// Mitsubishi GX Works2 project: mc_protocol   PLC: Q03UDV

PROGRAM MAIN
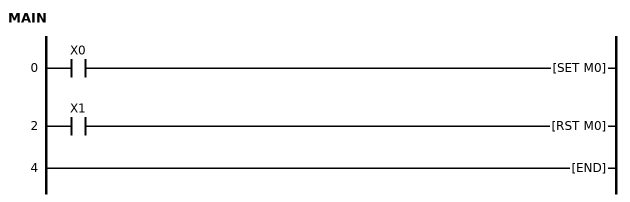
0     LD      X0
      SET     M0
2     LD      X1
      RST     M0
4     END
END_PROGRAM
